// Mitsubishi GX Works2 project: exam_q2   PLC: Q02/Q02H

PROGRAM exam_q2
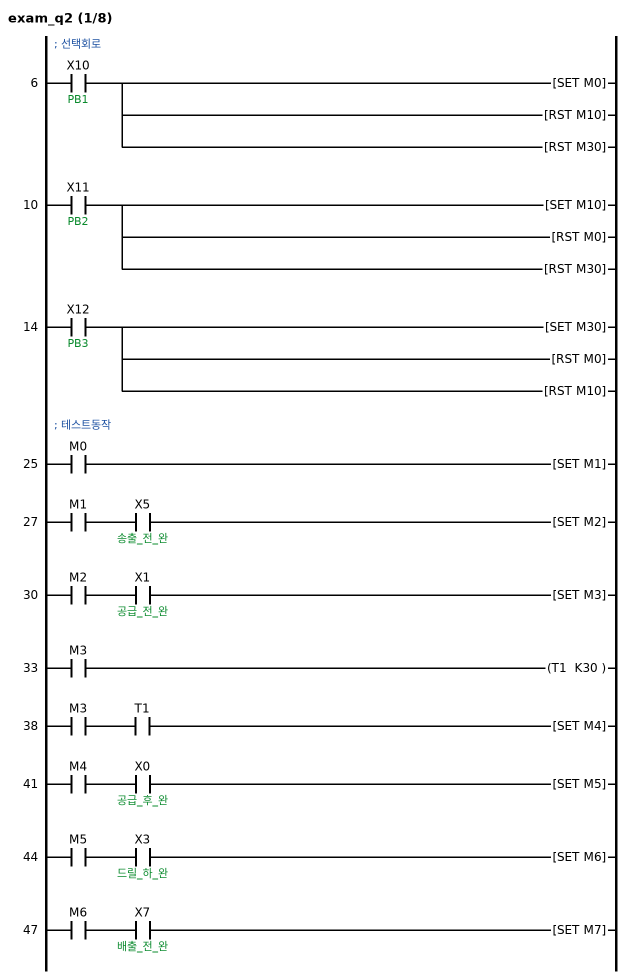
; 선택회로
6     LD      X10  ; PB1
      SET     M0
      RST     M10
      RST     M30
10    LD      X11  ; PB2
      SET     M10
      RST     M0
      RST     M30
14    LD      X12  ; PB3
      SET     M30
      RST     M0
      RST     M10
; 테스트동작
25    LD      M0
      SET     M1
27    LD      M1
      AND     X5  ; 송출_전_완
      SET     M2
30    LD      M2
      AND     X1  ; 공급_전_완
      SET     M3
33    LD      M3
      OUT     T1 K30
38    LD      M3
      AND     T1
      SET     M4
41    LD      M4
      AND     X0  ; 공급_후_완
      SET     M5
44    LD      M5
      AND     X3  ; 드릴_하_완
      SET     M6
47    LD      M6
      AND     X7  ; 배출_전_완
      SET     M7
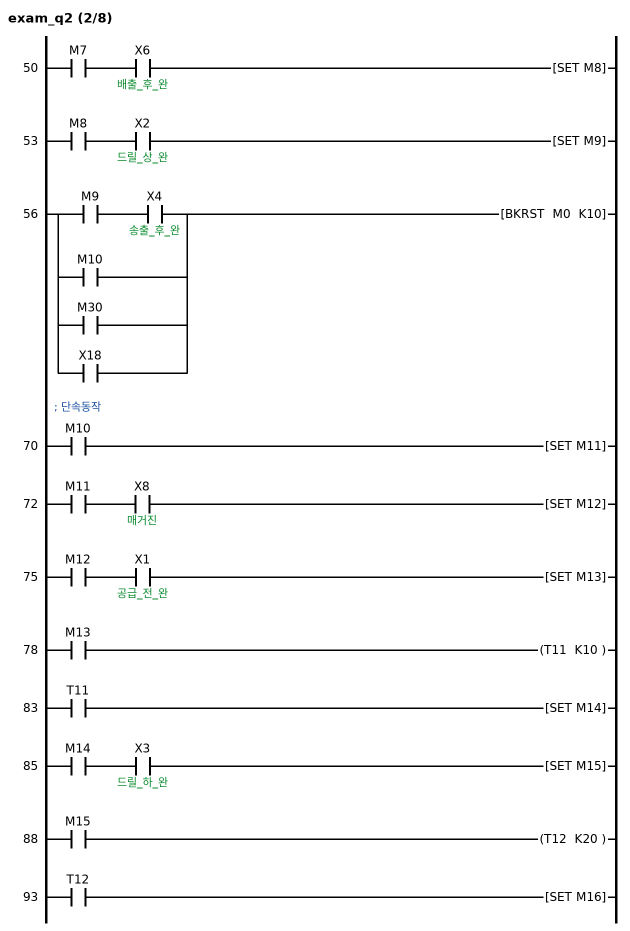
50    LD      M7
      AND     X6  ; 배출_후_완
      SET     M8
53    LD      M8
      AND     X2  ; 드릴_상_완
      SET     M9
56    LD      M9
      AND     X4  ; 송출_후_완
      OR      M10
      OR      M30
      OR      X18
      BKRST   M0 K10
; 단속동작
70    LD      M10
      SET     M11
72    LD      M11
      AND     X8  ; 매거진
      SET     M12
75    LD      M12
      AND     X1  ; 공급_전_완
      SET     M13
78    LD      M13
      OUT     T11 K10
83    LD      T11
      SET     M14
85    LD      M14
      AND     X3  ; 드릴_하_완
      SET     M15
88    LD      M15
      OUT     T12 K20
93    LD      T12
      SET     M16
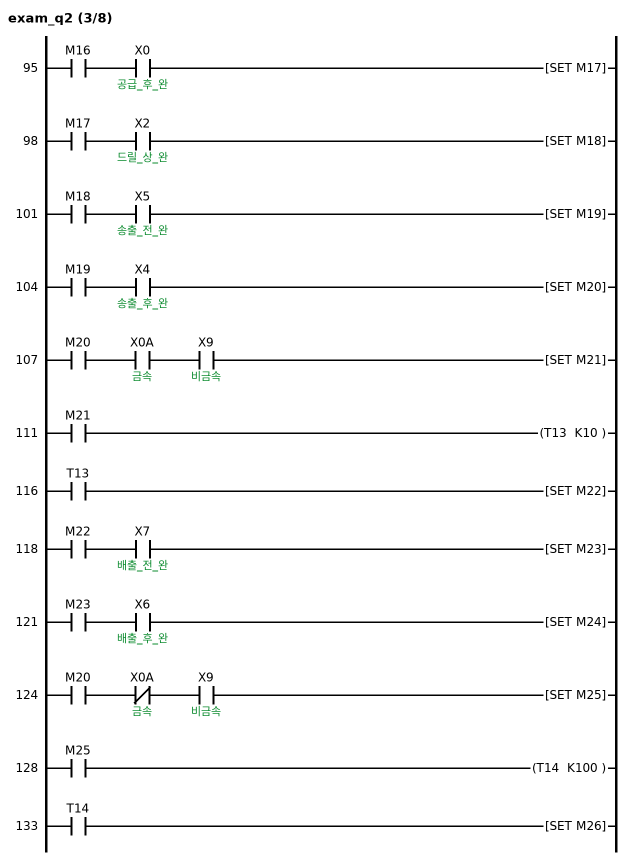
95    LD      M16
      AND     X0  ; 공급_후_완
      SET     M17
98    LD      M17
      AND     X2  ; 드릴_상_완
      SET     M18
101   LD      M18
      AND     X5  ; 송출_전_완
      SET     M19
104   LD      M19
      AND     X4  ; 송출_후_완
      SET     M20
107   LD      M20
      AND     X0A  ; 금속
      AND     X9  ; 비금속
      SET     M21
111   LD      M21
      OUT     T13 K10
116   LD      T13
      SET     M22
118   LD      M22
      AND     X7  ; 배출_전_완
      SET     M23
121   LD      M23
      AND     X6  ; 배출_후_완
      SET     M24
124   LD      M20
      ANI     X0A  ; 금속
      AND     X9  ; 비금속
      SET     M25
128   LD      M25
      OUT     T14 K100
133   LD      T14
      SET     M26
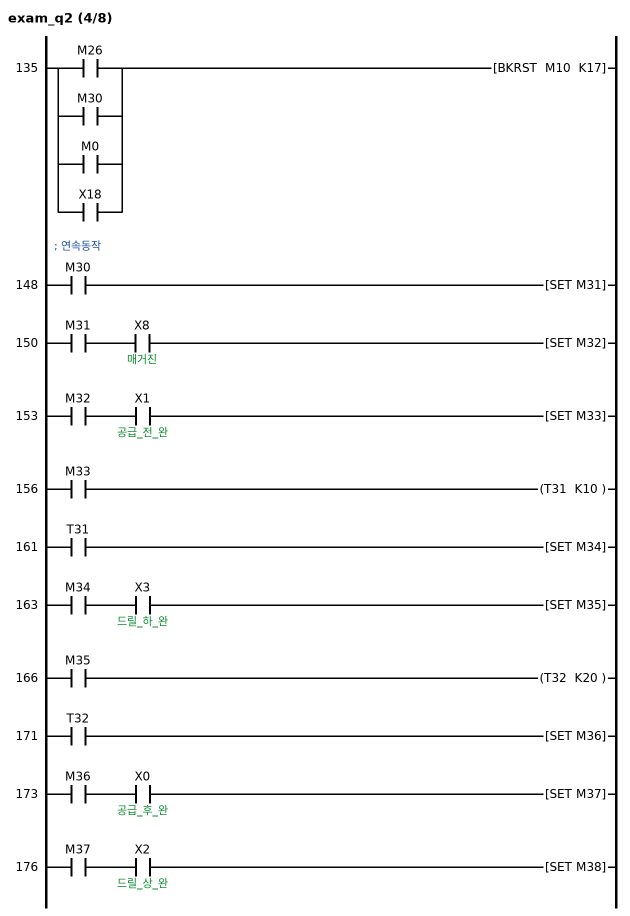
135   LD      M26
      OR      M30
      OR      M0
      OR      X18
      BKRST   M10 K17
; 연속동작
148   LD      M30
      SET     M31
150   LD      M31
      AND     X8  ; 매거진
      SET     M32
153   LD      M32
      AND     X1  ; 공급_전_완
      SET     M33
156   LD      M33
      OUT     T31 K10
161   LD      T31
      SET     M34
163   LD      M34
      AND     X3  ; 드릴_하_완
      SET     M35
166   LD      M35
      OUT     T32 K20
171   LD      T32
      SET     M36
173   LD      M36
      AND     X0  ; 공급_후_완
      SET     M37
176   LD      M37
      AND     X2  ; 드릴_상_완
      SET     M38
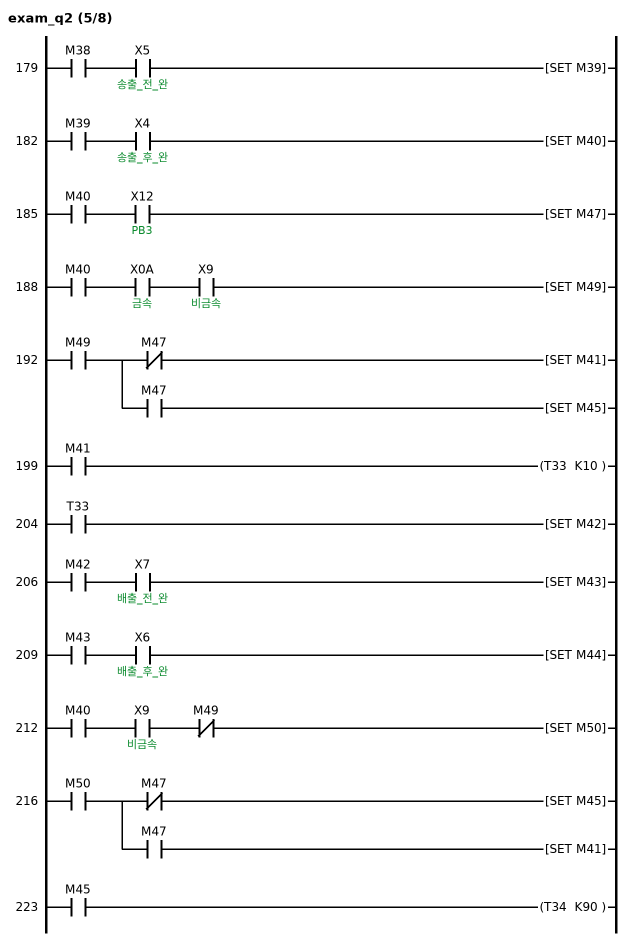
179   LD      M38
      AND     X5  ; 송출_전_완
      SET     M39
182   LD      M39
      AND     X4  ; 송출_후_완
      SET     M40
185   LD      M40
      AND     X12  ; PB3
      SET     M47
188   LD      M40
      AND     X0A  ; 금속
      AND     X9  ; 비금속
      SET     M49
192   LD      M49
      MPS
      ANI     M47
      SET     M41
      MPP
      AND     M47
      SET     M45
199   LD      M41
      OUT     T33 K10
204   LD      T33
      SET     M42
206   LD      M42
      AND     X7  ; 배출_전_완
      SET     M43
209   LD      M43
      AND     X6  ; 배출_후_완
      SET     M44
212   LD      M40
      AND     X9  ; 비금속
      ANI     M49
      SET     M50
216   LD      M50
      MPS
      ANI     M47
      SET     M45
      MPP
      AND     M47
      SET     M41
223   LD      M45
      OUT     T34 K90
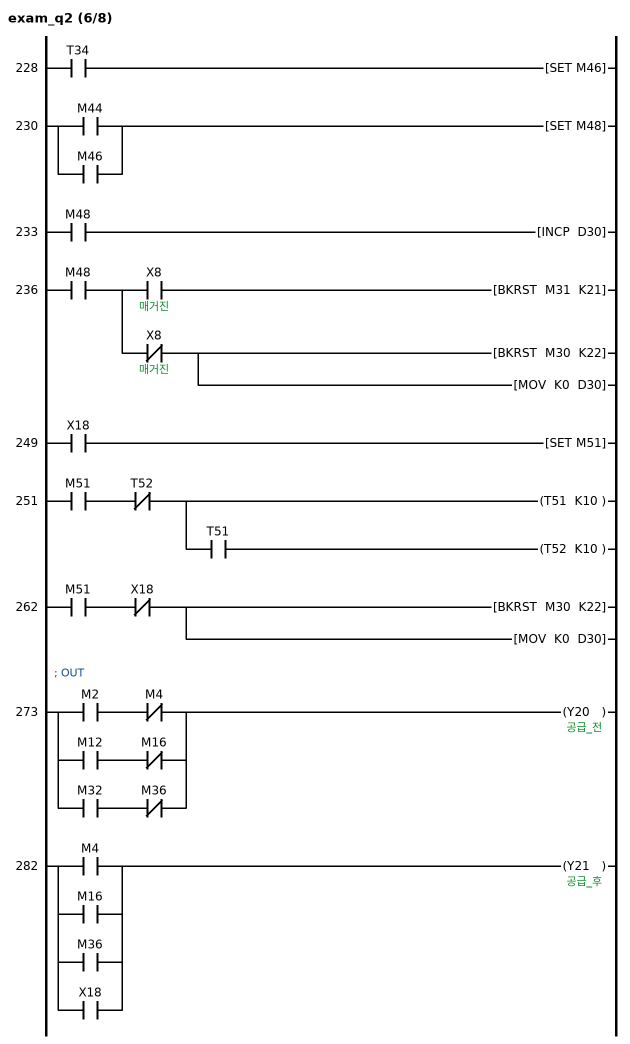
228   LD      T34
      SET     M46
230   LD      M44
      OR      M46
      SET     M48
233   LD      M48
      INCP    D30
236   LD      M48
      MPS
      AND     X8  ; 매거진
      BKRST   M31 K21
      MPP
      ANI     X8  ; 매거진
      BKRST   M30 K22
      MOV     K0 D30
249   LD      X18
      SET     M51
251   LD      M51
      ANI     T52
      OUT     T51 K10
      AND     T51
      OUT     T52 K10
262   LD      M51
      ANI     X18
      BKRST   M30 K22
      MOV     K0 D30
; OUT
273   LD      M2
      ANI     M4
      LD      M12
      ANI     M16
      ORB
      LD      M32
      ANI     M36
      ORB
      OUT     Y20  ; 공급_전
282   LD      M4
      OR      M16
      OR      M36
      OR      X18
      OUT     Y21  ; 공급_후
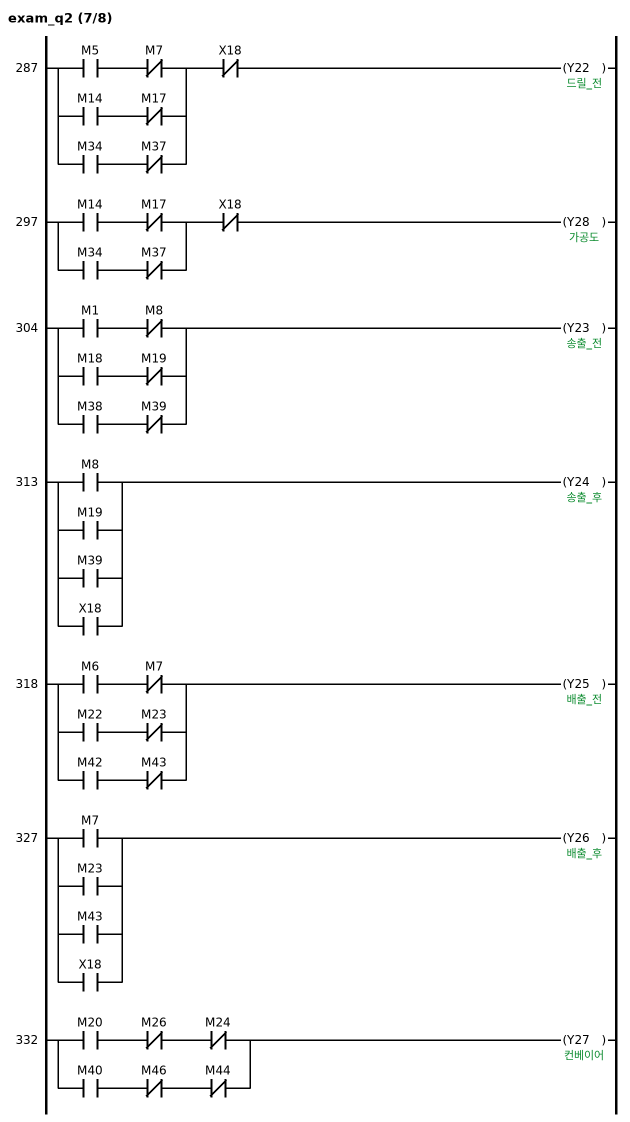
287   LD      M5
      ANI     M7
      LD      M14
      ANI     M17
      ORB
      LD      M34
      ANI     M37
      ORB
      ANI     X18
      OUT     Y22  ; 드릴_전
297   LD      M14
      ANI     M17
      LD      M34
      ANI     M37
      ORB
      ANI     X18
      OUT     Y28  ; 가공도
304   LD      M1
      ANI     M8
      LD      M18
      ANI     M19
      ORB
      LD      M38
      ANI     M39
      ORB
      OUT     Y23  ; 송출_전
313   LD      M8
      OR      M19
      OR      M39
      OR      X18
      OUT     Y24  ; 송출_후
318   LD      M6
      ANI     M7
      LD      M22
      ANI     M23
      ORB
      LD      M42
      ANI     M43
      ORB
      OUT     Y25  ; 배출_전
327   LD      M7
      OR      M23
      OR      M43
      OR      X18
      OUT     Y26  ; 배출_후
332   LD      M20
      ANI     M26
      ANI     M24
      LD      M40
      ANI     M46
      ANI     M44
      ORB
      OUT     Y27  ; 컨베이어
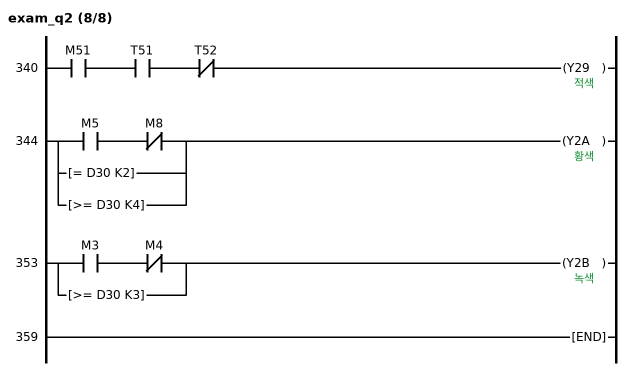
340   LD      M51
      AND     T51
      ANI     T52
      OUT     Y29  ; 적색
344   LD      M5
      ANI     M8
      OR=     D30 K2
      OR>=    D30 K4
      OUT     Y2A  ; 황색
353   LD      M3
      ANI     M4
      OR>=    D30 K3
      OUT     Y2B  ; 녹색
359   END
END_PROGRAM
